Staubli VAL3: constantes.dtx

mdesc mNomSpeed
public num nDRV_ACTIV
public num nRdy2SwitchON
public num nSwitchONDis
public num nNotRdySwiON
public num nSwitchedON
public num nOperatEnabled
public num nQuickStopActiv
public num nFaultReacActiv
public num nFaultState
public num nDRV_FAULT
num nEtapeInit
public num nNOTEXIST
public num nAXIS7
public num nAXIS8 = 1
public num nDEBUGDRIVE = 1
public num nHWALM_TESTHW
public num nHWALM_FEEDPW
public num nHWALM_UDRVOLT
public num nHWALM_OVRVOLT
public num nHWALM_OVRCUR
public num nHWALM_TEMPDIS
public num nHWALM_FRENO
public num nHWALM_EEPROM
public num nHWALM_FUSE5VLT
public num nHWALM_THERMMOT
public num nHWALM_HALL
public num nHWALM_TRANSDUC
public num nHWALM_CONNMOT
public num nSWALM_FUNGO
public num nSWALM_TAGLIA
public num nSWALM_CSDATI
public num nSWALM_I2T
public num nSWALM_POSITION
public num nSWALM_ENCODER
public num nSWALM_HALLENC
public num nSWALM_OVRSPEED
public num nSWALM_TRANSDUC
public num nSWALM_ENCMASTR
public num nSWALM_UDRVOLT
public num nSWALM_POSROTOR
public num nSWALM_OFFSREF
public num nSWALM_I2TREGEN
public num nSWALM_CANBUS
public num nSTATUS_REMOTE
public num nHOMINGMODE = 6
public num nINTERPMODE = 7
public num nTO_DRVENABLE
public num nTO_DRVDISABLE
public num nPPMODE
